(*
Nazwa:		FB_Gate
Opis:		Szlaban, siłownik
Wersja:		V0.1
Data:		22.05.2024
Autor:		DP
Urządzenia:	Jeden siłownik
Ostatnie zmiany:
	- RRRR-MM-DD [KTO?] Tekst Tekst Tekst Tekst Tekst Tekst Tekst Tekst Tekst Tekst 

Konfiguracja:
	- Krokówka
	Instukcja:
		-
		-
		-
	
Info:
	- Obsługa tylko jednego siłownika

*)

FUNCTION_BLOCK FB_Gate
VAR_INPUT
	bEnable										: BOOL;				//Zezwolenie na pracę
	bEStop										: BOOL;				//Stop awaryjny włączony
	bRun										: BOOL;				//Rozkaz przeciagania
	bHoming										: BOOL;				//Zezwolenie na wykonanie bazowania i pozycjonowanie układu
	bHeightSet									: BOOL;				//Ustaw do pozycji
	bIgnoreError								: BOOL;				//Ignorowanie błędów 
	bReset										: BOOL;				//Reset błędu, jeśli jest w stanie "eError"
	bResetCycle									: BOOL;				//Reset cyklu
	bUpSensor									: BOOL;				//
	bDownSensor									: BOOL;				//
	
	bManualMovement								: BOOL;				//Zezwolenie na ruchy ręczne

	_ALARMINFO_									: BOOL;
	iStationIndex								: UDINT;
	sStationName								: WSTRING;
END_VAR

VAR_OUTPUT
	eState										: E_Station;
	eRunningState								: E_Barrier;			// Stan 
	bError										: BOOL;					// Błąd stacji
	udiErrorID									: UDINT;				// Nr blędu 
	sErrorDescription							: STRING(200);			// Opis błędu
	sErrorDescription2							: STRING(200);			// Opis błędu
	sErrorStationName							: STRING;				// Nazwa stacji
	udiStationID								: UDINT;				// Nr stacji

	bActuator									: BOOL;					
				
	
	bCycleDone									: BOOL;					//Sygnał zakończenia cyklu
	bCycleNotDone								: BOOL;
	bHomingDone									: BOOL;
	tCycleTime									: TIME;					//Czas cyklu
	//Dodatkowe	
	eRunningStateBeforeEStop					: E_Barrier;			//Stan przed E-Stopem	
	bWasErrorOrEstop							: BOOL;
	
END_VAR

VAR
	(*LastStates*)
	eLastState									: E_Station;						//Stan ogólny bloku
	eLastStateTemp								: E_Station;						//Stan ogólny bloku
	eLastRunningState							: E_Barrier;						//Stan podbloku
	eLastRunningStateTemp						: E_Barrier;						//Stan podbloku
	            		
	(*Control*)
	tonResetting								: TON;								//Czas resetu
	tonHoming									: TON;
	tonPreparingToReady							: TON;								//Czas potrzeby na przygotowanie osi
	rtResetCommands								: R_TRIG;                                    	
	rtResetCycle								: R_TRIG;
	tonEstopDelay								: TON;
	
	(*Statistics*)
	tonCycleTimer								: TON;								//Czas cyklu przeciągania	
	rtrigCycleTimerRead							: R_TRIG;

	(*Homing*)
	iHomingCase									: INT;
	
	(*Aborting*)
	iAbortingCase								: INT;
	                                    	
	(*Errors*)
	bStateError									: BOOL;
	bResetCycleOn								: BOOL;
	tonUpSensor									: TON;	
	tonDownSensor								: TON;		
	
	(*Running*)

	tonNotDragActuatorDelay						: TON;
	tonRunningDraging							: TON;
	
	(*Inne*)
	
	iTest: INT;
	iTest1: INT;
	
		//Zmienne od EVENTLOGGER
	bAlarmInit 						: BOOL := TRUE; 
	nAlarmNumerator					: INT;
	arfbAlarm						: ARRAY[0..19] OF  FB_TcAlarm;		//Tablica bloczków błędów
	fbSourceInfo 					: FB_TcSourceInfo;
	iSourceInfo						: I_TcSourceInfo;
	sAlarmTest						: STRING;
	//Koniec zmiennych od EVENTLOGGER
	
END_VAR
	
VAR_IN_OUT
	bManualActuator								: BOOL;		

END_VAR

Signals();
ResetAll();
ErrorHandling();
Control();
Limits();
Statistics();
aStationID();

(*Zapisywanie ostatniego stanu*)
IF eLastStateTemp<>eState THEN
	eLastState := eLastStateTemp;
END_IF
eLastStateTemp := eState;
IF eLastRunningStateTemp<>eRunningState THEN
	eLastRunningState := eLastRunningStateTemp;
END_IF
eLastRunningStateTemp := eRunningState;
(*Koniec Zapisywanie ostatniego stanu*)

ACTION aStationID:
udiStationID	:=	iStationIndex;
END_ACTION

ACTION Control:
	(*****Wyłączenie enable*****)
	IF NOT bEnable AND NOT bError THEN
		IF eState <> E_Station.eDisabled AND eState <> E_Station.ePreparingToDisable THEN
				eState 								:= E_Station.ePreparingToDisable; 
		END_IF	
	END_IF

	(*****Estop*****)
	IF NOT bEstop  THEN	
		IF eState <> E_Station.eAborted AND eState <> E_Station.eAborting AND eState <> E_Station.eDisabled THEN
				eRunningStateBeforeEStop			:= eRunningState;
				eState 								:= E_Station.eAborting; 
				iAbortingCase						:= 0; 
		END_IF
	END_IF


	
CASE eState OF
	
//==========================================================================================	
	E_Station.eDisabled: 						// Stan nieaktywnosci (Stacja wyłączona) 
		
		IF bEnable THEN
			eState 									:= E_Station.ePreparingToReady; 
		END_IF 

//==========================================================================================	    
	E_Station.eAborted: 						// Stan bezpiecznego zatrzymania (po Abortingu) 	
			
		IF bEStop THEN
			bWasErrorOrEstop						:= TRUE;	
			eState 									:= E_Station.ePreparingToReady;
		END_IF		
			
//==========================================================================================	
	E_Station.eAborting:                 		// Stan bezpiecznego zatrzymywania (po EStopie)
		
		CASE iAbortingCase OF
			
			0: //Inicjalizacja
				iAbortingCase						:= 10;
				                                	
			10: //                              	
				iAbortingCase						:= 20;
		                                        	
			20: //Kasowanie komend              	
				//ResetCommands();                					                                                  	
				bManualActuator						:=	FALSE;		                                                      																			
				bResetCycleOn						:=	FALSE;					
				iHomingCase							:=	0;														
 				iAbortingCase						:=	40;
                                               	
			30: //Wyłączenie osi                	
				iAbortingCase						:= 30;
				                                	
			40: //Kasowanie podzespołow         	
				ResetCommands();                	
				iAbortingCase						:= 50;
				                                	
			50: //Przejście do Aborted          	
				iAbortingCase						:= 0;
				eState								:= E_Station.eAborted;
				eRunningState						:= E_Barrier.eReady;
				
		END_CASE

//==========================================================================================			
	E_Station.eError:                 	 		// Stan błędu 	
		
		bWasErrorOrEstop							:= TRUE;

		IF bReset THEN
			eState									:= E_Station.eResetting;	
		ELSE
			ResetCommands();
		END_IF
			
//==========================================================================================
	E_Station.eResetting:						// Stan resetowania bledu (po Errorze)
			
	//Procedura obsługi resetu w zależności od błędu
//	CASE (udiErrorID - iStationIndex) OF 
	bActuator							:= FALSE;		
// 	CASE udiErrorID OF 
// 
// 		131://Error 1 - Błąd siłownika przeciągania
// 			bActuator							:= FALSE;			
// 			bError								:= FALSE;	
// 			iTest :=	iTest	+	1;
// 		132://Error 2 - Błąd siłownika przeciągania
// 			bActuator							:= FALSE;			
// 			bError								:= FALSE;		
// 	
// 	END_CASE
	iTest1 :=	iTest1	+	1;
	
	IF NOT bError THEN
		udiErrorID									:= 0;
		sErrorDescription							:= '';
		sErrorDescription2							:= '';	
		eState										:= E_Station.ePreparingToReady;
	ELSIF tonResetting.Q THEN                   	
		eState										:= E_Station.eError;
	END_IF	
 
//==========================================================================================
	E_Station.eManualMovement:     				// Stan ruchów manualnych  
       
		ManualMovements();
		//Wyjście z trybu serwisowego
		IF NOT bManualMovement THEN
			bActuator								:=	bManualActuator;	
			eState									:=	E_Station.eReady;
		END_IF 

//==========================================================================================		
	E_Station.eHoming:							// Stan bazowania 
		
		Homing();	
		IF NOT bHoming AND NOT bHeightSet AND tonHoming.Q THEN
			eState									:=	E_Station.ePreparingToReady;
		END_IF		
			
//==========================================================================================
	E_Station.eHomingDone:                  	// Stan wykonania bazowania 

		bHomingDone									:= TRUE;
		bResetCycleOn								:= FALSE;		
		IF NOT bHoming AND NOT bHeightSet AND NOT bResetCycleOn THEN
		//	eState									:=	E_Station.eReady;
			eState									:=	E_Station.ePreparingToReady;
		END_IF

//==========================================================================================
	E_Station.ePreparingToReady:            	// Stan przygotowywania do gotowosci (zawsze przed Ready)  

		IF tonPreparingToReady.Q THEN
							
				ResetCommands();
				eState								:= E_Station.eReady;
				eRunningState						:= E_Barrier.eReady;
				
				IF bResetCycleOn THEN
					eState							:= E_Station.eHoming;
				END_IF
				
		END_IF			

//==========================================================================================
	E_Station.ePreparingToDisable:         	 	// Stan przygotowywania do nieaktywnosci (po wyłączeniu Enable) 
		
		bWasErrorOrEstop							:= FALSE;
		bHomingDone									:= FALSE;	
		
		ResetCommands();
		eState										:=	E_Station.eDisabled;
		eRunningState								:=	E_Barrier.eReady;


//==========================================================================================	
	E_Station.eReady:							// Stan gotowosci 


		(*Skasowanie wszystkich komend*)
		IF rtResetCommands.Q THEN	ResetCommands();	END_IF		
	
		IF bRun  (*AND NOT bCycleDone*) THEN
			eState									:= E_Station.eStarting;
		END_IF		
		IF bHoming OR bHeightSet THEN
			eState									:= E_Station.eHoming;
		END_IF
		IF bManualMovement THEN
			bManualActuator							:=	bActuator;							
			eState									:=	E_Station.eManualMovement;					
		END_IF
		IF NOT bRun THEN
			bCycleDone								:= FALSE;
		END_IF

//==========================================================================================
	E_Station.eStopping:					// Stan zatrzymywania 
		
		Running();
		IF eRunningState = E_Barrier.eReady THEN
			eState 									:= E_Station.eReady;
		END_IF


//==========================================================================================
	E_Station.eStarting:                  	// Stan uruchamiania (po Ready)
			
		eState										:= E_Station.eRunning;

//==========================================================================================
	E_Station.eRunning:               		// Stan wykonywania cyklu (po Startingu), w tym stanie osobny
 
		Running();

		IF NOT bRun  THEN					(*Przerywanie cyklu*)
			eState 				 					:= E_Station.eStopping;	
		END_IF
			
		//IF bCycleDone THEN (*Cykl zakończony*)
		//	eState 				 					:= E_Station.eReady;
		//END_IF	
		
//==========================================================================================
END_CASE
END_ACTION

ACTION ErrorHandling:
// Alarm_0200	200	Error	Siłownik | Blokada wysunięcia - sprawdź czujnik lub odblokuj
// Alarm_0201	201	Error	Siłownik | Blokada wsunięcia - sprawdź czujnik lub odblokuj
IF bAlarmInit THEN
    bAlarmInit := FALSE; 
	fbSourceInfo.Clear();
	fbSourceInfo.sName:=wsLiteral_TO_UTF8(sStationName);//'Machine';
	fbSourceInfo.nId:=udiStationID;//2700;
	// Alarm_0200	200	Error	Siłownik | Blokada wysunięcia - sprawdź czujnik lub odblokuj
    arfbAlarm[0].CreateEx(stEventEntry := TC_EVENTS.AlarmClass.Alarm_0200, bWithConfirmation:= FALSE,  ipSourceInfo:= fbSourceInfo); 
	// Alarm_0201	201	Error	Siłownik | Blokada wsunięcia - sprawdź czujnik lub odblokuj
	arfbAlarm[1].CreateEx(stEventEntry := TC_EVENTS.AlarmClass.Alarm_0201, bWithConfirmation:= FALSE,  ipSourceInfo:= fbSourceInfo);
END_IF



//CZYTANIE STATUSÓW
tonEstopDelay			(IN:=bEStop,	PT:=T#3S);
bStateError				:= (eState=E_Station.eError) OR (eState=E_Station.eResetting) OR NOT bEstop OR bIgnoreError;
//bStateError				:= (eState=E_Station.eError) OR (eState=E_Station.eResetting) OR bIgnoreError;

IF bEnable AND tonEstopDelay.Q THEN


	// Alarm_0200	200	Error	Siłownik | Blokada wysunięcia - sprawdź czujnik lub odblokuj
	//Error 1 - Błąd siłownika 
	tonDownSensor	(IN:= bActuator AND NOT bDownSensor	, PT:=T#2S);
	IF tonDownSensor.Q THEN
		IF NOT arfbAlarm[0].bActive THEN
			arfbAlarm[0].Raise(nTimeStamp:=0);
		END_IF
	ELSE	
		IF  arfbAlarm[0].bActive AND bReset THEN
			arfbAlarm[0].Clear(nTimeStamp:=0, bResetConfirmation:= FALSE);
		END_IF	
// 		bError								:= TRUE;
// 		udiErrorID							:= 131;	
// 		//udiErrorID 							:= udiErrorID + iStationIndex;
// 		sErrorDescription					:= 'Siłownik';
// 		sErrorDescription2					:= 'Blokada wysunięcia - sprawdź czujnik lub odblokuj';
	END_IF
	// Alarm_0201	201	Error	Siłownik | Blokada wsunięcia - sprawdź czujnik lub odblokuj
	//Error 2 - Błąd siłownika
	tonUpSensor	(IN:= NOT bActuator AND NOT bUpSensor	, PT:=T#2S);
	IF tonUpSensor.Q THEN
		IF NOT arfbAlarm[1].bActive THEN
			arfbAlarm[1].Raise(nTimeStamp:=0);
		END_IF
	ELSE	
		IF  arfbAlarm[1].bActive AND bReset THEN
			arfbAlarm[1].Clear(nTimeStamp:=0, bResetConfirmation:= FALSE);
		END_IF	

	END_IF;			
		
ELSE
	bError := FALSE;
END_IF

//******************PRZEJŚCIE DO eERROR*****************************

IF bError AND  NOT bStateError THEN
	eState 									:= E_Station.eError;
END_IF

//****************WYŚWIETLANIE STATUSU BLEDU************************
(*Wyświetlanie błedu na wyjściu*)
bError							:= FALSE;
FOR nAlarmNumerator := 0 TO 19 DO
	bError						:= bError OR arfbAlarm[nAlarmNumerator].bActive;
END_FOR

(*Przepisywanie nazwy stacji*)
sErrorStationName 							:= WSTRING_TO_STRING(sStationName);
END_ACTION

ACTION Homing:


IF bHoming THEN // Bazowanie - podjazd do góry i ustawienie obrotu
	CASE iHomingCase OF
	
	0: //
		bHomingDone										:= FALSE;		                                        		
		bActuator										:= FALSE;			
		iHomingCase										:= 10;
	
	10: //
		iHomingCase										:= 20;

	20: //
		iHomingCase										:= 30;
		
	30: //k
		iHomingCase										:= 40;
		
	40: //
		iHomingCase										:= 50;
	
	50: 
		iHomingCase										:= 60;
		
	60: //
		iHomingCase										:= 70;
			
	70:                             	
		iHomingCase										:= 80;

	80:
		iHomingCase										:= 100;
		
	100: //
		iHomingCase										:= 0;
		eState											:= E_Station.eHomingDone;
	
	END_CASE
END_IF	
IF bHeightSet THEN
	bActuator									:= FALSE;	
	eState										:= E_Station.eHomingDone;
END_IF
END_ACTION

ACTION Limits:
(*Wywowyłanie na początku*)


(*Prędkość zakręcania*)


(*Inny parametr*)
//...
END_ACTION

ACTION ManualMovements:

IF NOT bRun AND bManualMovement THEN                        	                                  	                                   	
	bActuator										:=	bManualActuator;			

ELSE
	bManualActuator									:=	FALSE;		
END_IF
	
IF bHoming THEN	
	eState											:=	E_Station.eHoming;	
END_IF                                                	
                                                      	
Running();

IF NOT bRun  THEN
	bCycleDone 										:= FALSE;
	bCycleNotDone 									:= FALSE;	
END_IF
END_ACTION

ACTION ResetAll:
(*****Reset bloczka*****)
IF bEnable THEN
	IF eState <> E_Station.eDisabled AND eState <> E_Station.ePreparingToDisable THEN
		IF bResetCycle THEN
			bResetCycleOn						:= TRUE;
			eState								:= E_Station.ePreparingToReady;
		END_IF
	END_IF
END_IF


IF bResetCycleOn THEN
	
	ResetCommands();
	eRunningState							:= E_Barrier.eReady;	
	eState 				 					:= E_Station.eReady;

END_IF
END_ACTION

ACTION ResetCommands:
//KAsowanie komend ruchu 
                                                     	
bManualActuator											:=	FALSE;		                                                      	
bActuator												:=	FALSE;	
                                                    	
bResetCycleOn											:=	FALSE;	

iHomingCase												:=	0;
//bCycleDone								   				:=	FALSE;
END_ACTION

ACTION Running:
	
CASE eRunningState OF
	
	E_Barrier.eDisabled:
		eRunningState								:= E_Barrier.eReady; 
	
	E_Barrier.eReady:

		//IF NOT bCycleDone  THEN                                           	
			IF bRun THEN   
				bActuator								:=	FALSE;
				eRunningState							:=	E_Barrier.eWaitingToOpen; 
       		END_IF
		//END_IF
		
	E_Barrier.eWaitingToOpen:
	
		bActuator										:=	TRUE;
		IF bDownSensor THEN
			eRunningState								:=	E_Barrier.eOpen; 
		END_IF
	
	E_Barrier.eOpen:	
		bCycleDone										:= TRUE;	
		eRunningState									:= E_Barrier.eDone;	
	
	E_Barrier.eDone:			
		
		IF NOT bRun THEN
			eRunningState								:=	E_Barrier.eWaitingToClose; 
		END_IF
		
	E_Barrier.eWaitingToClose:
	
		bActuator										:=	FALSE;
		IF bUpSensor THEN
			eRunningState								:=	E_Barrier.eReady; 
		END_IF
	

		
END_CASE
END_ACTION

ACTION Signals:

tonPreparingToReady		(IN:=	eState = E_Station.ePreparingToReady			,PT:= T#3S);
tonResetting			(IN:=	eState = E_Station.eResetting					,PT:= T#200MS);
tonHoming				(IN:=	eState = E_Station.eHoming						,PT:= T#1S);
rtResetCommands			(CLK:=	eState = E_Station.eReady 						,Q=>);
END_ACTION

ACTION Statistics:
rtrigCycleTimerRead(CLK:=bCycleDone);
IF rtrigCycleTimerRead.Q THEN
	tCycleTime:=tonCycleTimer.ET;
END_IF
tonCycleTimer(IN:= eRunningState>E_Barrier.eReady, PT:=T#1D);
END_ACTION

END_FUNCTION_BLOCK

(* stored: Version 1.1.0.1, ProductVersion 3.1.4026.13, FileIdentifier deb689510705b5b71fa3fab0cdd797c5d4bbdfb0, FileSignature 6993ce1f1d97c4708842ac908977a2d695472d715fd8cf67cf7ae9f98d70fd9ab9b8e34e39e419b7510cd69759849e1955553b1369289170ddceac6ec7da0ae62cfbd75a119e6b50dbb9aa2bf35c353edb0d50a8775324c5399a48acadc24a5de745e6e3da7669c35f685b1550573473cd1a38efc93275c413f0acb22f9f01e62213a955570d00d9ff9168a8cefe642b7d05a2f8ffde3599088048998599416d0f63a7c7134f1404c317931a2b740dc51b9859f1cc0cd16fb7117f203b91de637a60ad32d2b38f3da6288ac0ec4c31e645e37fa3c36ba7fceeeac395ab99fc3637bad8b959cffc8e448ef0c7665e222c68032868970787a5e9a2345f3654da80
   POU FB_Gate: Id {51db0df5-0da6-46f0-b3ea-1d0c72adcce1}, SpecialFunc None
   Action aStationID: Id {c9fa46a9-3361-4d05-baf0-506c4551ac1a}
   Action Control: Id {2caa1aa4-4aa9-42de-87f3-7940a12a80f0}
   Action ErrorHandling: Id {25b04d25-024a-48d5-b4b6-f0aee2fcad53}
   Action Homing: Id {8f50612a-03e1-4a08-beb6-c49e394a2252}
   Action Limits: Id {2147077d-e893-4f56-b23c-05e2fac057ae}
   Action ManualMovements: Id {9d1b5247-10cd-419f-8ecd-b5b99de53274}
   Action ResetAll: Id {938d24d2-9158-42a9-9f30-3d25ea40be27}
   Action ResetCommands: Id {f55ec511-b165-4879-9a80-15fdaf91b19c}
   Action Running: Id {fcd9be5a-9af2-448d-a064-8164e995c260}
   Action Signals: Id {f72f89fb-e5db-4073-94a4-783324266194}
   Action Statistics: Id {247505de-f901-4ff5-b50e-7804a9bae9c2} *)
